Fanuc KAREL source: kf00053.KL

-- PROVISIONAL review KL for V770-1; original PC SHA256 b4b65208b9c11c5f2efdd5870de34dbd6706af32e50a591eae734bf52858716b
-- Incomplete behavior may be omitted. Consult companion uncertainty JSON. Do not deploy.
PROGRAM KF00053
%NOLOCKGROUP
VAR
  I : INTEGER
  J : INTEGER
  X : REAL
  Y : REAL
  B : BOOLEAN
  C : BOOLEAN
  TXT : STRING[80]
  TXT2 : STRING[80]
  STATUS : INTEGER
-- UNRESOLVED_DECL AI type=002010
-- UNRESOLVED_DECL BI type=002010
-- UNRESOLVED_DECL P type=000102
-- UNRESOLVED_DECL JP type=000199
-- UNRESOLVED_DECL PF type=000101
-- UNRESOLVED_DECL V1 type=000013
-- UNRESOLVED_DECL V2 type=000013
BEGIN
  -- UNRESOLVED_PC offsets 5-12; opcodes 9C,23
  -- UNRESOLVED_PC offsets 22-36; opcodes 21,9D,52,23
  -- UNRESOLVED_PC offsets 41-58; opcodes 21,2E,5C,79
  -- UNRESOLVED_PC offsets 63-67; opcodes 7F
END KF00053
